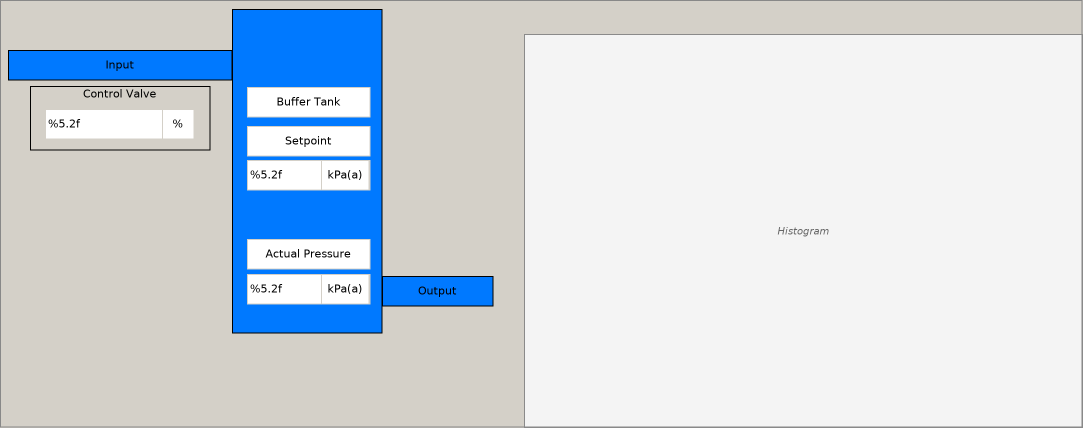
VISUALIZATION Tank_Visualization  // 1083x428
    RoundedRectangle (30,86 180x64), "Control Valve"
    RoundedRectangle (232,9 150x324)
    Rectangle (382,276 111x30), "Output"
    Rectangle (8,50 224x30), "Input"
    Textfield (247,87 123x30), "Buffer Tank"
    Textfield (45,109 150x30), "%5.2f", text variable: Input_Control_Valve.HMI_Valve_Reference
    Textfield (247,274 123x30), "%5.2f", text variable: Tank_Pressure.Input_SI
    Textfield (321,274 48x30), "kPa(a)"
    Textfield (162,109 32x30), "%"
    Textfield (247,160 123x30), "%5.2f", text variable: Input_Control_Valve.Controller_Setpoint
    Textfield (321,160 48x30), "kPa(a)"
    Textfield (247,126 123x30), "Setpoint"
    Textfield (247,239 123x30), "Actual Pressure"
    Histogram (524,34 559x394), scale format: %.1f, scale 0..500
END_VISUALIZATION

(* stored: Version 1.1.0.1, ProductVersion 3.1.4024.15
   Visu Tank_Visualization: Id {eeca4abf-6641-4415-94f1-f734d0995b86} *)
